{attribute 'qualified_only'}
{attribute 'strict'}
{attribute 'to_string'}
TYPE E_InletToSystem :
(
	Recirculation_From_Storage:=1,Hydrogen_Inlet:=2
);
END_TYPE

(* stored: Version 1.1.0.1
   DUT E_InletToSystem: Id {68df0664-ec30-4823-8cf2-8238beee26db} *)
